Staubli VAL3: MotionQueue.pjx

--- MotionQueue.pjx ---
Parameters version=s7.7.2 stackSize=5000 millimeterUnit=true
Program file=clear.pgx
Program file=pop.pgx
Program file=push.pgx
Program file=start.pgx
Program file=stop.pgx
Data file=MotionQueue.dtx
Type name=MotionBuffer path=Disk://ros_libs/MotionBuffer/MotionBuffer.pjx

--- MotionQueue.dtx ---
num nPush
num nPop
public num nElems
MotionBuffer buffer[10]
  [0]
    mdesc mDesc = {leave=0, reach=0}
    num nDuration
    num nSequence
    jointRx jJointRx
  [1]
    mdesc mDesc = {leave=0, reach=0}
    num nDuration
    num nSequence
    jointRx jJointRx
  [2]
    mdesc mDesc = {leave=0, reach=0}
    num nDuration
    num nSequence
    jointRx jJointRx
  [3]
    mdesc mDesc = {leave=0, reach=0}
    num nDuration
    num nSequence
    jointRx jJointRx
  [4]
    mdesc mDesc = {leave=0, reach=0}
    num nDuration
    num nSequence
    jointRx jJointRx
  [5]
    mdesc mDesc = {leave=0, reach=0}
    num nDuration
    num nSequence
    jointRx jJointRx
  [6]
    mdesc mDesc = {leave=0, reach=0}
    num nDuration
    num nSequence
    jointRx jJointRx
  [7]
    mdesc mDesc = {leave=0, reach=0}
    num nDuration
    num nSequence
    jointRx jJointRx
  [8]
    mdesc mDesc = {leave=0, reach=0}
    num nDuration
    num nSequence
    jointRx jJointRx
  [9]
    mdesc mDesc = {leave=0, reach=0}
    num nDuration
    num nSequence
    jointRx jJointRx

--- getNumElements.pgx ---
public program getNumElements(num& x_nNumElems)
begin
  x_nNumElems = nElems
end
